RESOURCE_TYPE ResourceType1
  (* Standard: 61499-2 *)
  (* Version 0.1, 2016-00-15, Hammond, HAMMONDSDESKTOP *)
  VAR_INPUT
    Variable1 : BOOL;
  END_VAR
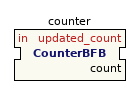
  FBS
    counter : CounterBFB;
  END_FBS
END_RESOURCE_TYPE
